Fanuc KAREL source: kd00009.KL

-- PROVISIONAL review KL for V1013-1; original PC SHA256 96fe1c68bfdfaf7c765e64e44dc7a4dfb03b4de84f760cf709f2d0e7a7509193
-- Incomplete behavior may be omitted. Consult companion uncertainty JSON. Do not deploy.
PROGRAM KD00009
%NOLOCKGROUP
VAR
  I : INTEGER
  J : INTEGER
  B : BOOLEAN
  R : REAL
  S : STRING[80]
BEGIN
  -- UNRESOLVED_PC offsets 5-12; opcodes 9D,23
  -- UNRESOLVED_PC offsets 17-21; opcodes 7F
END KD00009
